// TwinCAT 3 PLC project plcProject
// ProgramVersion: 3.1.4024.0
// libraries:
//   Tc2_ModbusSrv, * (Beckhoff Automation GmbH)
//   Tc2_Standard, * (Beckhoff Automation GmbH)
//   Tc2_SUPS, * (Beckhoff Automation GmbH)
//   Tc2_System, * (Beckhoff Automation GmbH)
//   Tc2_Utilities, * (Beckhoff Automation GmbH)
//   Tc3_Module, * (Beckhoff Automation GmbH)
//   Util, * (System)
// project tree:
//   DUTs/ Word2real.TcDUT, DEVICE.TcDUT, PF_ET.TcDUT, READ_PAR.TcDUT, WRITE_PAR.TcDUT
//   GVLs/ GVL.TcGVL
//   / PlcTask.TcTTO
//   POUs/ FB_READ_WITHOUT_TIMER.TcPOU, MAIN.TcPOU
// real-time tasks:
//   TASK PlcTask: cycle T#10ms, priority 20, ADS port 350

CONFIGURATION plcProject
    RESOURCE PLC ON TwinCAT3
        TASK PlcTask(INTERVAL := T#10ms, PRIORITY := 20);
        PROGRAM MAIN WITH PlcTask : MAIN;
    END_RESOURCE
END_CONFIGURATION

// ---- DUTs/Word2real.TcDUT
TYPE Word2real :
UNION
	var1 : ARRAY [1..2] OF WORD;	//Be carefull of position, var[1] is LSB, var[2]MSB
	var2 : REAL;
	var3: ARRAY[1..4] OF BYTE;
END_UNION
END_TYPE

// ---- DUTs/DEVICE.TcDUT
TYPE DEVICE :
STRUCT
	//CONFIGURATION PARAMETER FB READ
	ID: STRING(15);
	ServerIP: STRING(15);
	ServerNumPort: UINT;
	ServerReadUnitID: BYTE;
	
	//ReadBusy: BOOL;
	//ReadError: BOOL;
	
	//INVERTER VALUE WRITE
	
	//ServerWriteUnitID: BYTE;
	//ReactivePowerSetPoint :INT;
	//ActivePowerSetPoint : INT;
	//PowerFactorSetPoint :INT;
	//PowerFactorExcitationType : DINT;
	
	
	readTimestamp : UDINT; 
	readParameterCounter : INT := 0;
	readParameter : ARRAY[1..GVL.MAX_READ_PARAMETER] OF READ_PAR;
	
	CheckComm: UDINT;
	
	//writeParameter : ARRAY[1..GVL.MAX_READ_PARAMETER] OF WRITE_PAR;
	
END_STRUCT
END_TYPE

// ---- DUTs/PF_ET.TcDUT
TYPE PF_ET :
STRUCT
	A: ARRAY[1..2] OF WORD;
END_STRUCT
END_TYPE

// ---- DUTs/READ_PAR.TcDUT
TYPE READ_PAR :
STRUCT
	id : DINT := 0;
	ReadAddress: WORD := 0;
	ReadQty: WORD := 0;
	ModbusFunction : BYTE := 0;
	ReadCount: WORD;
 
	AuxArr : ARRAY[1..GVL.MAX_VALUE_FOR_READ_PARAMETER] OF WORD;
	
	//fault : BOOL := FALSE;
	//TypeArr : ARRAY[1..GVL.MAX_VALUE_FOR_READ_PARAMETER] OF STRING;
	//ValueArr: ARRAY[1..GVL.MAX_VALUE_FOR_READ_PARAMETER] OF REAL;
	
	bBusy: BOOL;
	bError: BOOL;
	
END_STRUCT
END_TYPE

// ---- DUTs/WRITE_PAR.TcDUT
TYPE WRITE_PAR :
STRUCT
	WriteAddress: WORD;
	WriteQty: WORD;
	AuxArr : ARRAY[1..10] OF DINT;
	
	bBusy: BOOL;
	bError: BOOL;
	commTrig: R_TRIG;
END_STRUCT
END_TYPE

// ---- GVLs/GVL.TcGVL
VAR_GLOBAL CONSTANT
	MAX_DEVICE : UINT := 32 + 16; //32
	MAX_READ_PARAMETER : INT := 128 + 128 ; //128
	MAX_VALUE_FOR_READ_PARAMETER : INT := 128 + 128; //128;
	
	
	MAX_IO : UINT := 32 + 32 ;
  
	//testEAP AT %Q*: BYTE;

END_VAR

VAR_GLOBAL 
	
	devices: ARRAY[1..MAX_DEVICE] OF DEVICE;
	devicesCount: INT;
	
	primaryTime : TIME := T#15S;  

	PLC_On: BOOL := FALSE;

	mb_Output_Registers : ARRAY [1..MAX_IO] OF WORD;
	
	enableRTU : BOOL := FALSE;
	enableIO : BOOL := FALSE;
	
END_VAR

// ---- POUs/MAIN.TcPOU
PROGRAM MAIN
VAR
	fbRead: ARRAY [1..GVL.MAX_DEVICE] OF FB_READ_WITHOUT_TIMER;
	
	start : BOOL := TRUE;

	//delay : TIME := T#10MS;
	
	tTime : TIME;  
	currentTime : TIME := TIME();
	  
	//bExecute : BOOL := FALSE;
	timermodbus: TON;
	
	//inpArray AT %I* : ARRAY[1..GVL.MAX_IO, 1..16] OF BOOL ;
	
	
END_VAR

ParallelScan();
//SerialScan();
//IOScan();


METHOD IOScan : BOOL

VAR
	//i : INT;
	//j : INT;
END_VAR

(*
IF GVL.enableIO THEN
	FOR i := 1 TO GVL.MAX_IO DO
		GVL.mb_Output_Registers[i]  := 0;
		
		FOR j := 1 TO 16 DO
		   IF  inpArray[i, j] THEN
			   GVL.mb_Output_Registers[i] := GVL.mb_Output_Registers[i]  + LREAL_TO_WORD(EXPT( 2, j - 1 ));
		   END_IF
		END_FOR;
	END_FOR
END_IF
*)
END_METHOD

METHOD ParallelScan : BOOL
VAR_INPUT
END_VAR

VAR
	

	i: INT := 0;
	testCount : ULINT := 0;
	
END_VAR
IF GVL.PLC_On AND GVL.devicesCount > 0  THEN
		
	timermodbus(IN:= NOT timermodbus.Q, PT:= GVL.primaryTime, Q=> , ET=> );
		
	i := 1;
	
	WHILE ( i <= GVL.devicesCount ) DO
		
		IF timermodbus.Q THEN
			testCount := testCount + 1;
			
			tTime := TIME() - currentTime;
			currentTime := TIME();
		END_IF; 
		
		IF GVL.devices[ i ].ServerIP <> '' THEN  
		
			fbRead[ i ](
				device := GVL.devices[ i ],
				bExecute := timermodbus.Q
			);	
		END_IF
		
		i := i + 1;
	END_WHILE

END_IF
END_METHOD

METHOD SerialScan : BOOL
VAR_INPUT
END_VAR

VAR
	i: INT := 0;
	testCount : ULINT := 0;

	timermodbusRTU: TON;
	
	subState: INT;	
	execRead : BOOL;
	
END_VAR
END_METHOD

END_PROGRAM

// ---- POUs/FB_READ_WITHOUT_TIMER.TcPOU
FUNCTION_BLOCK FB_READ_WITHOUT_TIMER

VAR_IN_OUT
	device: DEVICE;
	bExecute : BOOL;
END_VAR

VAR_OUTPUT
	execRead : BOOL := FALSE;
END_VAR

VAR
	
	fbTime   : FB_LocalSystemTime := ( bEnable := TRUE, dwCycle := 1 );
	
	readInputRegister : FB_MBReadInputRegs;
	readHoldingRegister : FB_MBReadRegs;
	

	//TYPE_ARR: ARRAY[1..2] OF STRING; 
	done: BOOL;
	
	timeOut: TIME := T#2S;
	readError : INT := 0;
	idError : UDINT;
	
	k: UINT;
	z: INT;
	
	switch_first_bit: INT;
	Aux_Dword: DWORD;
	
	j: INT := 0;
	
	timer: TON;
	delay : TIME := T#200MS;
	
	index : INT := 0;
	subState: INT;
	
	ReadInputs: INT;
END_VAR

	
IF bExecute AND NOT execRead THEN
	execRead 			:= TRUE;
	index 				:= 1;
	subState 			:= 6;
	
	readError 			:= 0;
	idError 			:= 0;
	
	device.CheckComm 	:= 0;

	fbTime();
	device.readTimestamp := DT_TO_UDINT( SYSTEMTIME_TO_DT( fbTime.systemTime ) );
END_IF



IF execRead THEN
	
	CASE subState OF
		
		1: 
			IF device.readParameter[index].id <> 0 THEN 
				
				subState := 2;
				
				IF device.readParameter[index].ModbusFunction = 3 THEN	
				
					readHoldingRegister(
						sIPAddr:= device.ServerIP, 
						nTCPPort:= device.ServerNumPort, 
						nUnitID:= device.ServerReadUnitID, 
						nQuantity:= device.readParameter[index].ReadQty, 
						nMBAddr:= device.readParameter[index].ReadAddress, 
						cbLength:= SIZEOF(WORD) * device.readParameter[index].ReadQty, 
						pDestAddr:= ADR(device.readParameter[index].AuxArr), 
						bExecute:= TRUE , 
						tTimeout:= timeOut, 
						bBusy=> device.readParameter[index].bBusy, 
						bError=>,
						(*bBusy=> device.ReadBusy,
						bError => device.ReadError,*)
						nErrId=>, 
						cbRead=> 
					);	
					
						

				ELSIF device.readParameter[index].ModbusFunction = 4 THEN
					
					
					readInputRegister(
						sIPAddr:= device.ServerIP, 
						nTCPPort:= device.ServerNumPort, 
						nUnitID:= device.ServerReadUnitID, 
						nQuantity:= device.readParameter[index].ReadQty, 
						nMBAddr:= device.readParameter[index].ReadAddress, 
						cbLength:= SIZEOF(WORD) * device.readParameter[index].ReadQty, 
						pDestAddr:= ADR(device.readParameter[index].AuxArr), 
						bExecute:= TRUE ,  
						tTimeout:= timeOut, 
						bBusy=> device.readParameter[index].bBusy, 
						bError=>,
						(*bBusy=> device.ReadBusy,
						bError => device.ReadError,*)
						nErrId=>, 
						cbRead=> 
					);
				
					
					
				END_IF
			ELSE
				subState := 3;
			END_IF
			
		2: 
			
			IF device.readParameter[index].ModbusFunction = 3 THEN
				
				IF readHoldingRegister.bError THEN
 					IF readHoldingRegister.nErrId = 1861 THEN
						idError := idError +1 ;
					END_IF
					
					device.CheckComm := readHoldingRegister.nErrId;
					
					device.readParameter[index].bError := TRUE; 
					subState := 4;
				ELSIF NOT readHoldingRegister.bBusy THEN
					
					device.readParameter[index].bError := FALSE;
					subState := 4;
				END_IF
				
			
				readHoldingRegister(bExecute:= FALSE);
			
				
				
			ELSIF device.readParameter[index].ModbusFunction = 4 THEN
				
				IF readInputRegister.bError THEN
					
					IF readInputRegister.nErrId = 1861 THEN
						idError := idError +1 ;
					END_IF
					
					device.CheckComm := readInputRegister.nErrId;
					
					device.readParameter[index].bError := TRUE;
					subState := 4;
				
				ELSIF NOT readInputRegister.bBusy THEN
					device.readParameter[index].bError := FALSE;
					subState := 4;
				END_IF
   
				readInputRegister(bExecute:= FALSE);
				
			END_IF
						
			
		3: 
			// EXIT
			execRead := FALSE; 
			
		4: // INCREMENT
			timer(IN:= NOT timer.Q, PT:= delay, Q=> , ET=> );
			
			IF timer.Q THEN
				index := index + 1;
				subState := 6;
			END_IF
			
		6: 	// CHECK
			IF index > device.readParameterCounter THEN
				subState := 3;
			ELSE 
				subState := 1;
			END_IF
		
		ELSE
			// Azioni di default se nessun altro caso corrisponde
			//errore := TRUE;
			execRead := FALSE;
			
	END_CASE;
END_IF

END_FUNCTION_BLOCK
